TYPE
    ST_WheelhouseInput :
    STRUCT
        WheelhouseA : ST_WheelhouseTour;
        WheelhouseB : ST_WheelhouseTour;
    END_STRUCT
END_TYPE

(* stored: Version 1.1.0.1, ProductVersion 3.1.4024.13
   DUT ST_WheelhouseInput: Id {2cb46f4c-e12a-4d53-82cd-7194de9e30f0} *)
